PROGRAM P_Serial_Com
VAR
	fbSerialLineControl_EL6001_M1K3: SerialLineControl;
	fbSerialLineControl_EL6001_M2K3: SerialLineControl;
END_VAR

//These are the global IOs...don't forget to copy your data into them

(* EL6001 Serial port 0 com function *)
fbSerialLineControl_EL6001_M1K3(Mode:= SERIALLINEMODE_EL6_22B (*SERIALLINEMODE_KL6_22B_STANDARD*),
						        pComIn:= ADR(Serial_stComIn_M1K3),
						   	    pComOut:=ADR(Serial_stComOut_M1K3),
						        SizeComIn:= SIZEOF(Serial_stComIn_M1K3),
						        TxBuffer:= Serial_TXBuffer_M1K3,
						        RxBuffer:= Serial_RXBuffer_M1K3,
						        Error=> ,
						        ErrorID=> );

fbSerialLineControl_EL6001_M2K3(Mode:= SERIALLINEMODE_EL6_22B (*SERIALLINEMODE_KL6_22B_STANDARD*),
						        pComIn:= ADR(Serial_stComIn_M2K3),
						   	    pComOut:=ADR(Serial_stComOut_M2K3),
						        SizeComIn:= SIZEOF(Serial_stComIn_M2K3),
						        TxBuffer:= Serial_TXBuffer_M2K3,
						        RxBuffer:= Serial_RXBuffer_M2K3,
						        Error=> ,
						        ErrorID=> );

END_PROGRAM

(* stored: Version 1.1.0.1, ProductVersion 3.1.4022.18
   POU P_Serial_Com: Id {fa981f30-4d2c-4d48-ab6c-00ec78d696a1}, SpecialFunc None *)
